(*

.. <legal notes>

legal notes
=================
| SPDX-FileCopyrightText: © 2025 Oleksandr Tiutyk <trofimich@gmail.com>
| SPDX-License-Identifier: LGPL-3.0-only
| For details check: LGPL-3.0-only_

.. _LGPL-3.0-only: https://www.gnu.org/licenses/lgpl-3.0.en.html

.. </legal notes>

*)

INTERFACE IWaitAndPickActivity EXTENDS IActivity

METHOD AddBarnch : DINT
VAR_INPUT
	condition : ICondition;
	activity : IActivity;
END_VAR
END_METHOD

{attribute 'monitoring' := 'call'}
PROPERTY FINAL CurrentActivity : IActivity
GET
END_GET
END_PROPERTY

{attribute 'monitoring' := 'call'}
PROPERTY FINAL CurrentBranchIndex : DINT
GET
END_GET
END_PROPERTY

END_INTERFACE

(* stored: Version 1.1.0.1
   Itf IWaitAndPickActivity: Id {d4864be5-0eac-415d-b629-65950d177917}
   Method AddBarnch: Id {478ff588-0885-4c43-a728-aedd9396b880}
   Property CurrentActivity: Id {857432f2-2a97-4edb-9b8b-fa7ee28db595}
   Get Get: Id {40e9165a-2ec4-4875-8f14-88eddbd2971d}
   Property CurrentBranchIndex: Id {7a572bc2-ab06-4776-a888-8d0b4b9dd766}
   Get Get: Id {6b1b8141-bc92-48e4-a8ff-e1b2b063dfde} *)
